{attribute 'GeneratedUsingTerminal: EP6228-3132-0016'}
{attribute addProperty BoxType "EP6228-3132-0016"}
{attribute addProperty Id "Digital_InputsDigital_Inputs_3DEC2D274"}
{attribute addProperty CRC "916462649"}
{attribute addProperty Size "4"}
TYPE Module_11_Digital_Inputs_36A01C39 :
STRUCT
	{attribute addProperty Name "Digital_Inputs"}
	Digital_Inputs  : Digital_Inputs_3DEC2D27;
END_STRUCT
END_TYPE

(* stored: Version 1.2.0.0, ProductVersion 3.1.4024.9
   DUT Module_11_Digital_Inputs_36A01C39: Id {58c8ff54-57de-4df7-ae3b-8afb8f8f5384} *)
